FUNCTION_BLOCK INTERNAL FINAL FB_FooMessage IMPLEMENTS I_Message

(*
syntax = "proto3";

import "tchaxx-extensions.proto";

message Foo
{
  Bar bar = 1;
  repeated Baz baz = 2 [(tchaxx.ext.v1.array_length) = 3];
}

message Bar
{
  string name = 1;
  uint32 age = 2;
  optional string email = 3;
}

message Baz
{
  fixed32 value = 1;
  string name = 2;
}
*)

VAR
	fbMessageParser : FB_MessageParser(ipMessage:= THIS^);
    fbMessageWriter : FB_MessageWriter(ipMessage:= THIS^);	  
    fbBar           : FB_BarMessage;
    fbBaz           : FB_BazMessage;
    stFoo           : ST_Foo;
    nField2Index    : UDINT; 
END_VAR

// Repeated Fields
VAR
	fbRepeatedBazCodec	: FB_FieldCodecMessage(nTag:= 16#0A, ipMessage:= fbBaz);
	fbRepeatedBaz		: FB_RepeatedField(anyArray:= F_ToAnyType(stFoo.baz), anyFirstElem:= F_ToAnyType(stFoo.baz[0]));
END_VAR

{warning 'Add method implementation '}
(* Calculates the size of this message in Protocol Buffer wire format, in bytes.*)
METHOD CalculateSize : UDINT
END_METHOD

(* Merges the data from the specified coded input stream with the current message.*)
METHOD MergeFrom : HRESULT
VAR_IN_OUT
	fbParseCtx : FB_ParseContext;
END_VAR
VAR
    nTag : UDINT;
END_VAR
nField2Index := 0;

REPEAT   
MergeFrom := fbParseCtx.ReadTag(nTag=> nTag);
IF SUCCEEDED(MergeFrom) AND nTag = 0 THEN
    EXIT;
END_IF;

IF FAILED(MergeFrom) THEN
    RETURN;
END_IF

CASE nTag OF
    16#0A:         // Bar bar = 1;
    ;
         MergeFrom := fbParseCtx.ReadMessage(ipMessage:= fbBar);
         THIS^.stFoo.bar := fbBar.Bar;
         
    16#12:         // repeated Baz baz = 2 ;
        ;
           MergeFrom := fbRepeatedBaz.AddEntriesFrom(fbParseCtx:= fbParseCtx, ipFieldCodec:= fbRepeatedBazCodec);
ELSE
    MergeFrom := fbParseCtx.SkipLastField();
END_CASE

UNTIL (FAILED(MergeFrom) OR nTag = 0)
END_REPEAT
END_METHOD

PROPERTY MessageValue : T_Any
GET
MessageValue := F_ToAnyType(anyArg:= THIS^.stFoo);
END_GET
END_PROPERTY

PROPERTY PUBLIC Parser : REFERENCE TO FB_MessageParser
GET
Parser REF= THIS^.fbMessageParser;
END_GET
END_PROPERTY

(* Writer for this message.*)
PROPERTY Writer : REFERENCE TO FB_MessageWriter
GET
Writer REF= THIS^.fbMessageWriter;
END_GET
END_PROPERTY

(* Writes the data to the given coded output stream.*)
METHOD WriteTo : HRESULT
VAR_IN_OUT
	(* Coded output stream to write the data to. *)
	fbWriteCtx	: FB_WriteContext;
END_VAR

// fbWriteCtx.WriteRepeatedField(fbRepeatedBaz);

fbRepeatedBaz.WriteTo(fbWriteCtx, fbRepeatedBazCodec);

// fbWriteCtx.WriteRepeatedFieldMessage(iMessage:= fbBaz, F_ToAnyType(stFoo.baz), F_ToAnyType(stFoo.baz[0]), 3, nTag:= 16#12);
END_METHOD

END_FUNCTION_BLOCK

(* stored: Version 1.1.0.1
   POU FB_FooMessage: Id {cf2e5f3a-ec46-4558-9f26-acb076490d6c}, SpecialFunc None
   Method CalculateSize: Id {ce3905cf-bfcb-4319-9024-c4cd79291450}
   Method MergeFrom: Id {314e9c79-e00c-4e2b-9692-cca9b4200ec9}
   Property MessageValue: Id {cfd2a290-9591-4704-8795-fa192bf92b2c}
   Get Get: Id {730fa78a-e2c7-45ae-94f0-b57d65c6664f}
   Property Parser: Id {ae3443db-ae7b-4a70-9ffa-eae02af28c01}
   Get Get: Id {8bc398e2-c1c2-4f53-9cd1-8f8f69928cba}
   Property Writer: Id {9c398de1-5ca6-4b01-afe8-c1794cb882c7}
   Get Get: Id {b34af9f5-d7d6-48fc-8953-36329690d1ef}
   Method WriteTo: Id {43cf5782-5084-41c2-8543-7116a19d9763} *)
